{attribute 'qualified_only'}
{attribute 'strict'}
TYPE E_Step :
(
	// Special steps
	NoStep := -32767,	// No step
	Unknown := -32000,	// Unknown step
	
	// Not Enabled or Errors
	NeOrError := -990,	// Not enabled or at fault
	
	// Recovery
	Recovering := 990,	// Restore After Failure

	// Stopping
	Stopping := 900,	// Nominal shutdown
	
	// Stop
	Stop := 0, 			// Stop
	
	// Working steps
	Waiting	:= 100,		// Waiting for object
	Feeding := 200,		// Object Transfer
	Unloading := 300	// Outgoing object discharge
   
);
END_TYPE
//  NoStep = '-32767'
//  Unknown = '-32000'
//  NeOrError = '-990'

(* stored: Version 1.1.0.1, ProductVersion 3.1.4024.12
   EnumerationTextList E_Step: Id {55de7b00-de84-4f53-a951-c988b78497f3} *)
